# EPICS substitutions: apfelApp/Db/apfelHadcon.substitutions
file apfelHadcon.template {
pattern {
    protocolFile,
#   PREFIX,
    NAME, SUFFIX
}
	{ "hadcon_APFEL0.proto"
#     "PANDA:"
	  "APFEL" "" }
}
